(* IEC 61131-3 sources: Industry-PLC-LLM/data/PLCBEAD_repo/PLCBEAD_PLCEmbed-main/PLC-BEAD/Source/GEB/CEIL2, 1 file *)

(* ---- CEIL2.ST ---- *)
FUNCTION _REAL_TO_DINT:DINT
  VAR_INPUT
    X :	REAL;
  END_VAR

  IF REAL_TO_DINT(0.5) = DINT#1 THEN
    _REAL_TO_DINT := REAL_TO_DINT(X);
    RETURN;
  END_IF;

  IF X > 0.0 THEN
    _REAL_TO_DINT := REAL_TO_DINT(X+0.5);
  ELSIF X < 0.0 THEN
    _REAL_TO_DINT := REAL_TO_DINT(X-0.5);
  ELSE
    _REAL_TO_DINT := DINT#0;
  END_IF;
END_FUNCTION

FUNCTION CEIL2:DINT

	VAR_INPUT
		X :	REAL;
	END_VAR

	CEIL2 := _REAL_TO_DINT(X);
	IF DINT_TO_REAL(CEIL2) < X THEN
			CEIL2 := CEIL2 + DINT#1;
	END_IF;

END_FUNCTION

PROGRAM program0
  VAR
    LocalVar0 : REAL;
    CEIL5_OUT : DINT;
  END_VAR

  CEIL5_OUT := CEIL2(LocalVar0);
END_PROGRAM
